PROGRAM PRG_DiagnosticPaddleMotors
VAR
    fbDPX_Motor : FB_MotionStage;
    fbDPY_Motor : FB_MotionStage;
    fbDPZ_Motor : FB_MotionStage;
END_VAR

stDPXMotor.bPowerSelf := TRUE;
fbDPX_Motor(stMotionStage:=Main.stDPXMotor);

// Deal with bad limit switch on Y stage
stDPYMotor.bLimitBackwardEnable := TRUE;
stDPYMotor.bLimitForwardEnable := TRUE;
stDPYMotor.bPowerSelf := TRUE;
fbDPY_Motor(stMotionStage:=Main.stDPYMotor);

stDPZMotor.bPowerSelf := TRUE;
fbDPZ_Motor(stMotionStage:=Main.stDPZMotor);

END_PROGRAM

(* stored: Version 1.1.0.1, ProductVersion 3.1.4024.6
   POU PRG_DiagnosticPaddleMotors: Id {698f952c-e0c1-49b9-9654-83f2078781a3}, SpecialFunc None *)
